{attribute 'GeneratedUsingTerminal: EJ6910-0000-0018'}
{attribute addProperty BoxType "EJ6910-0000-0018"}
{attribute addProperty Id "FSLOGIC_InputsAT %I*FSLOGIC_Inputs_EEE9388E2FSLOGIC_OutputsAT %I*EMPTY_STRUCTURE0WcStateAT %I*WcState_9091E0EB2InfoDataAT %I*InfoData_32EB74EA10"}
{attribute addProperty CRC "3444433408"}
{attribute addProperty Size "14"}
TYPE EJ6910_CD4DE200 EXTENDS EtcSlaveTerminalBase_947E5A46 :
STRUCT
	{attribute addProperty Name "FSLOGIC_Inputs"}
	FSLOGIC_Inputs : FSLOGIC_Inputs_EEE9388E;
	{attribute addProperty Name "FSLOGIC_Outputs"}
	FSLOGIC_Outputs : EMPTY_STRUCTURE;
	{attribute addProperty Name "WcState"}
	WcState : WcState_9091E0EB;
	{attribute addProperty Name "InfoData"}
	InfoData : InfoData_32EB74EA;
END_STRUCT
END_TYPE

(* stored: Version 1.2.0.0, ProductVersion 3.1.4024.9
   DUT EJ6910_CD4DE200: Id {4823f113-a8bd-4428-b8b3-a7e2742955c0} *)
